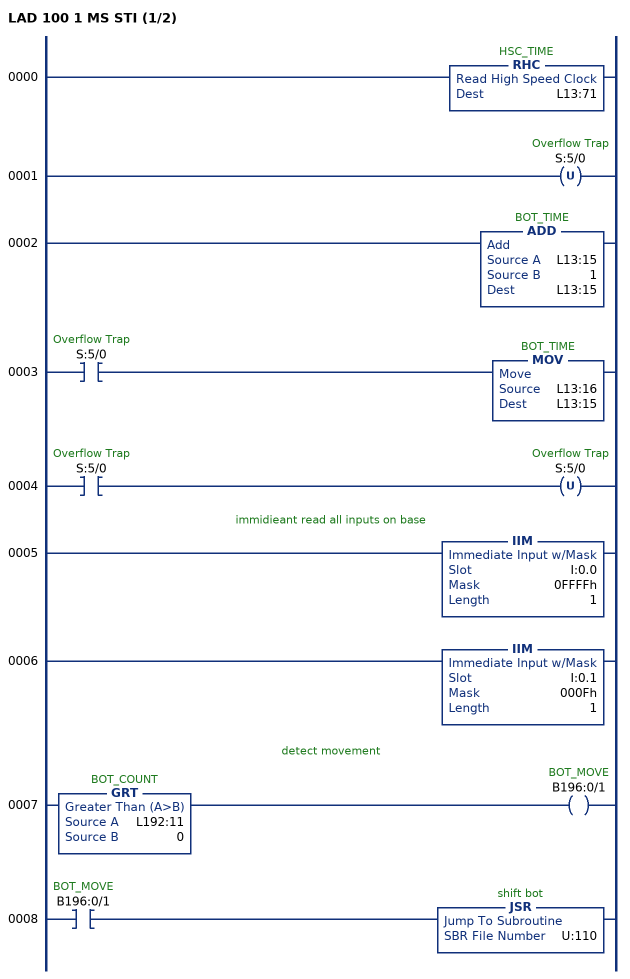
% Rung: 0 %
SOR RHC L13:71 EOR
%   L13:71  HSC_TIME %
% Rung: 1 %
SOR OTU S:5/0 EOR
%   S:5/0  "Overflow Trap" %
% Rung: 2 %
SOR ADD L13:15 1 L13:15 EOR
%   L13:15  BOT_TIME %
% Rung: 3 %
SOR XIC S:5/0 MOV L13:16 L13:15 EOR
%   S:5/0  "Overflow Trap" %
%   L13:16  MIN_LONG %
%   L13:15  BOT_TIME %
% Rung: 4 %
SOR XIC S:5/0 OTU S:5/0 EOR
%   S:5/0  "Overflow Trap" %
% Rung: 5 %
% immidieant read all inputs on base %
SOR IIM I:0.0 0FFFFh 1 EOR
% Rung: 6 %
SOR IIM I:0.1 000Fh 1 EOR
% Rung: 7 %
% detect movement %
SOR GRT L192:11 0 OTE B196:0/1 EOR
%   L192:11  BOT_COUNT %
%   B196:0/1  BOT_MOVE %
% Rung: 8 %
SOR XIC B196:0/1 JSR U:110 EOR
%   B196:0/1  BOT_MOVE %
%   U:110  "shift bot" %

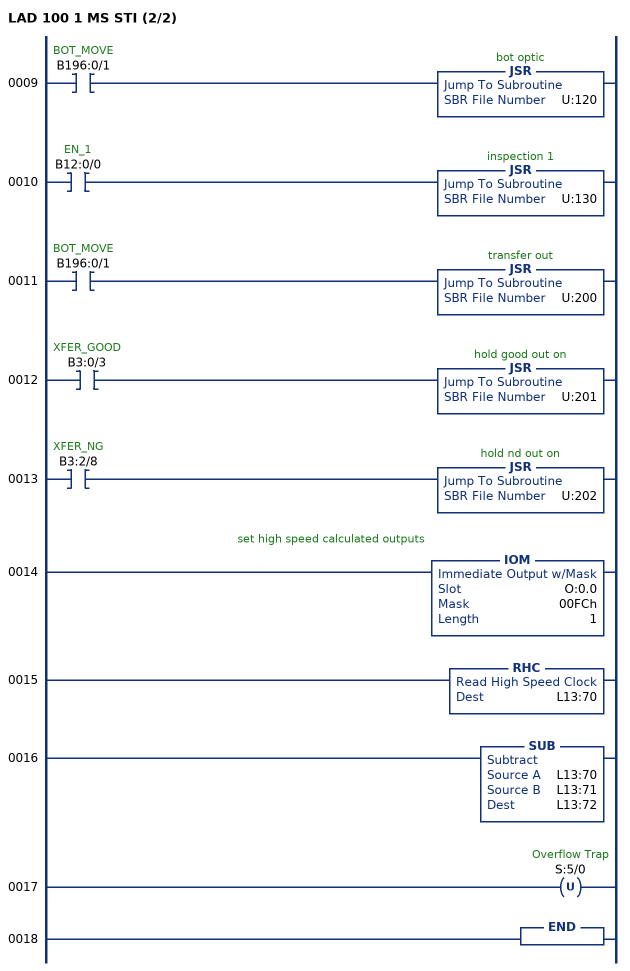
% Rung: 9 %
SOR XIC B196:0/1 JSR U:120 EOR
%   B196:0/1  BOT_MOVE %
%   U:120  "bot optic" %
% Rung: 10 %
SOR XIC B12:0/0 JSR U:130 EOR
%   B12:0/0  EN_1 %
%   U:130  "inspection 1" %
% Rung: 11 %
SOR XIC B196:0/1 JSR U:200 EOR
%   B196:0/1  BOT_MOVE %
%   U:200  "transfer out" %
% Rung: 12 %
SOR XIC B3:0/3 JSR U:201 EOR
%   B3:0/3  XFER_GOOD %
%   U:201  "hold good out on" %
% Rung: 13 %
SOR XIC B3:2/8 JSR U:202 EOR
%   B3:2/8  XFER_NG %
%   U:202  "hold nd out on" %
% Rung: 14 %
% set high speed calculated outputs %
SOR IOM O:0.0 00FCh 1 EOR
% Rung: 15 %
SOR RHC L13:70 EOR
% Rung: 16 %
SOR SUB L13:70 L13:71 L13:72 EOR
%   L13:71  HSC_TIME %
% Rung: 17 %
SOR OTU S:5/0 EOR
%   S:5/0  "Overflow Trap" %
% Rung: 18 %
SOR END EOR

LADDER 102 "SPEED BOT"    % high speed %
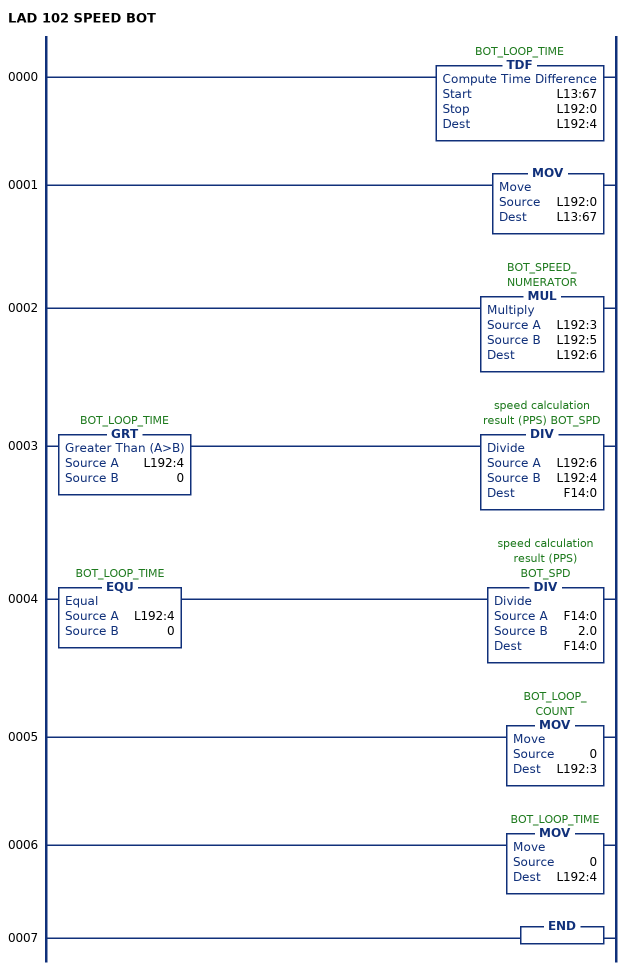
% Rung: 0 %
SOR TDF L13:67 L192:0 L192:4 EOR
%   L192:0  BOT_THIS_TIME  "rtc bot belt movement event time" %
%   L192:4  BOT_LOOP_TIME %
% Rung: 1 %
SOR MOV L192:0 L13:67 EOR
%   L192:0  BOT_THIS_TIME  "rtc bot belt movement event time" %
% Rung: 2 %
SOR MUL L192:3 L192:5 L192:6 EOR
%   L192:3  BOT_LOOP_COUNT %
%   L192:5  TKS_PER_SECOND %
%   L192:6  BOT_SPEED_NUMERATOR %
% Rung: 3 %
SOR GRT L192:4 0 DIV L192:6 L192:4 F14:0 EOR
%   L192:4  BOT_LOOP_TIME %
%   L192:6  BOT_SPEED_NUMERATOR %
%   F14:0  BOT_SPD  "speed calculation result (PPS)" %
% Rung: 4 %
SOR EQU L192:4 0 DIV F14:0 2.0 F14:0 EOR
%   L192:4  BOT_LOOP_TIME %
%   F14:0  BOT_SPD  "speed calculation result (PPS)" %
% Rung: 5 %
SOR MOV 0 L192:3 EOR
%   L192:3  BOT_LOOP_COUNT %
% Rung: 6 %
SOR MOV 0 L192:4 EOR
%   L192:4  BOT_LOOP_TIME %
% Rung: 7 %
SOR END EOR

LADDER 104 "P BOT"    % high speed %
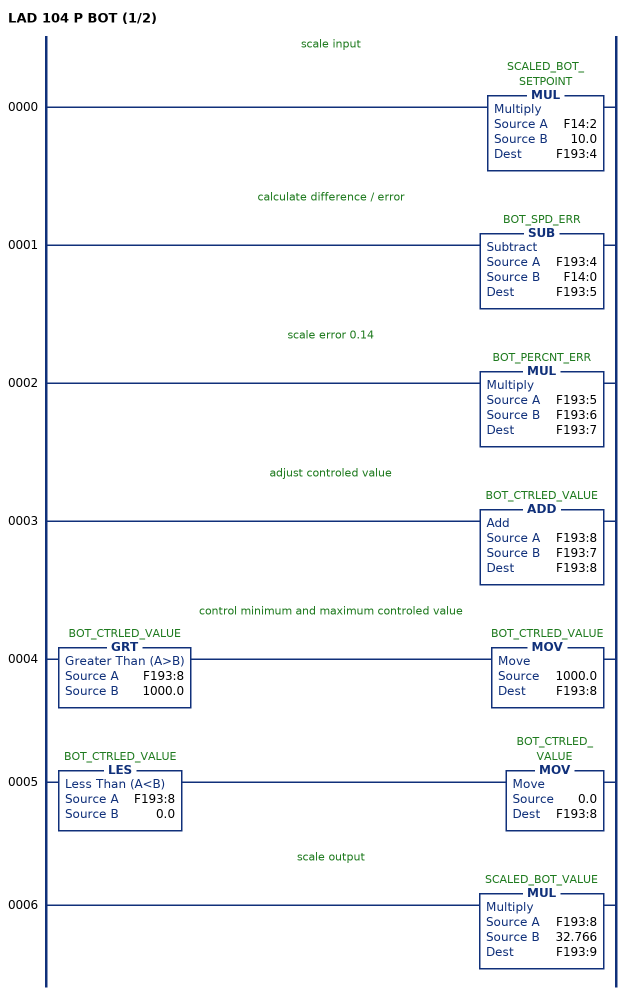
% Rung: 0 %
% scale input %
SOR MUL F14:2 10.0 F193:4 EOR
%   F14:2  BOT_SPD_SETPOINT %
%   F193:4  SCALED_BOT_SETPOINT %
% Rung: 1 %
% calculate difference / error %
SOR SUB F193:4 F14:0 F193:5 EOR
%   F193:4  SCALED_BOT_SETPOINT %
%   F14:0  BOT_SPD  "speed calculation result (PPS)" %
%   F193:5  BOT_SPD_ERR %
% Rung: 2 %
% scale error 0.14 %
SOR MUL F193:5 F193:6 F193:7 EOR
%   F193:5  BOT_SPD_ERR %
%   F193:6  BOT_FDBK_RATIO %
%   F193:7  BOT_PERCNT_ERR %
% Rung: 3 %
% adjust controled value %
SOR ADD F193:8 F193:7 F193:8 EOR
%   F193:8  BOT_CTRLED_VALUE %
%   F193:7  BOT_PERCNT_ERR %
% Rung: 4 %
% control minimum and maximum controled value %
SOR GRT F193:8 1000.0 MOV 1000.0 F193:8 EOR
%   F193:8  BOT_CTRLED_VALUE %
% Rung: 5 %
SOR LES F193:8 0.0 MOV 0.0 F193:8 EOR
%   F193:8  BOT_CTRLED_VALUE %
% Rung: 6 %
% scale output %
SOR MUL F193:8 32.766 F193:9 EOR
%   F193:8  BOT_CTRLED_VALUE %
%   F193:9  SCALED_BOT_VALUE %

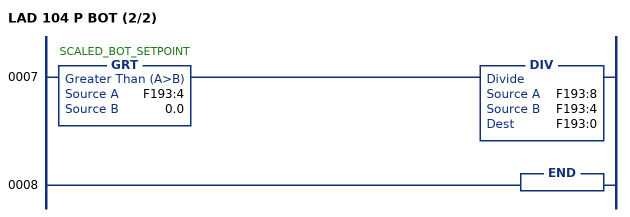
% Rung: 7 %
SOR GRT F193:4 0.0 DIV F193:8 F193:4 F193:0 EOR
%   F193:4  SCALED_BOT_SETPOINT %
%   F193:8  BOT_CTRLED_VALUE %
% Rung: 8 %
SOR END EOR

LADDER 110 "SHIFT BOT"
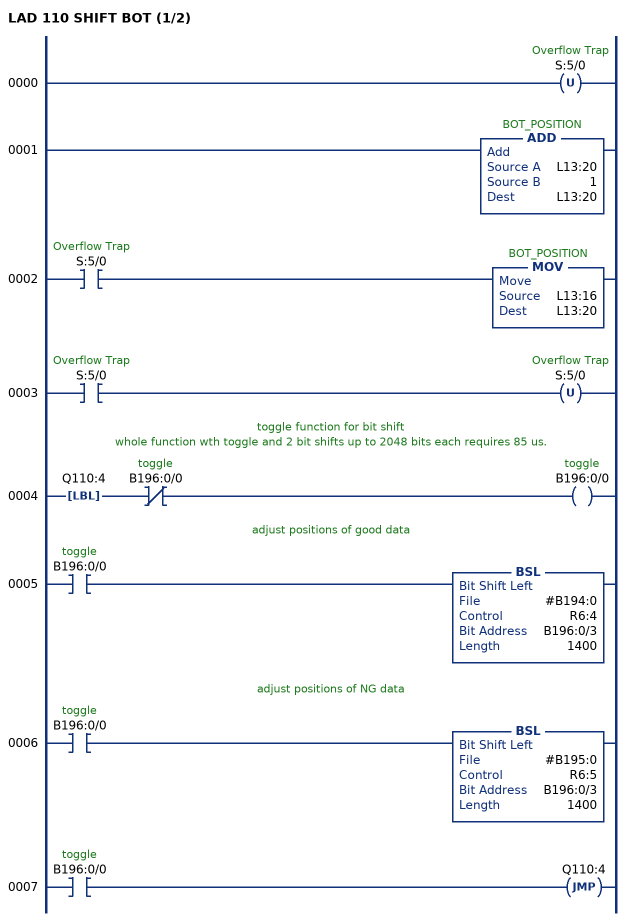
% Rung: 0 %
SOR OTU S:5/0 EOR
%   S:5/0  "Overflow Trap" %
% Rung: 1 %
SOR ADD L13:20 1 L13:20 EOR
%   L13:20  BOT_POSITION %
% Rung: 2 %
SOR XIC S:5/0 MOV L13:16 L13:20 EOR
%   S:5/0  "Overflow Trap" %
%   L13:16  MIN_LONG %
%   L13:20  BOT_POSITION %
% Rung: 3 %
SOR XIC S:5/0 OTU S:5/0 EOR
%   S:5/0  "Overflow Trap" %
% Rung: 4 %
% toggle function for bit shift
% whole function wth toggle and 2 bit shifts up to 2048 bits each requires 85 us. %
SOR LBL Q110:4 XIO B196:0/0 OTE B196:0/0 EOR
%   B196:0/0  "toggle" %
% Rung: 5 %
% adjust positions of good data %
SOR XIC B196:0/0 BSL #B194:0 R6:4 B196:0/3 1400 EOR
%   B196:0/0  "toggle" %
%   B196:0/3  OFF %
% Rung: 6 %
% adjust positions of NG data %
SOR XIC B196:0/0 BSL #B195:0 R6:5 B196:0/3 1400 EOR
%   B196:0/0  "toggle" %
%   B196:0/3  OFF %
% Rung: 7 %
SOR XIC B196:0/0 JMP Q110:4 EOR
%   B196:0/0  "toggle" %

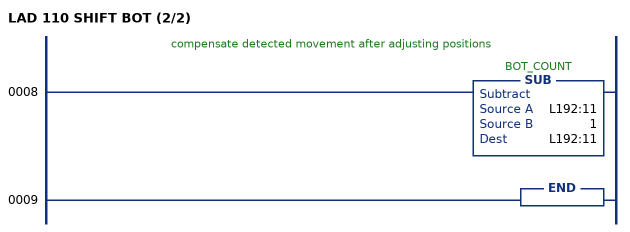
% Rung: 8 %
% compensate detected movement after adjusting positions %
SOR SUB L192:11 1 L192:11 EOR
%   L192:11  BOT_COUNT %
% Rung: 9 %
SOR END EOR

LADDER 120 "BOTOPTIC"
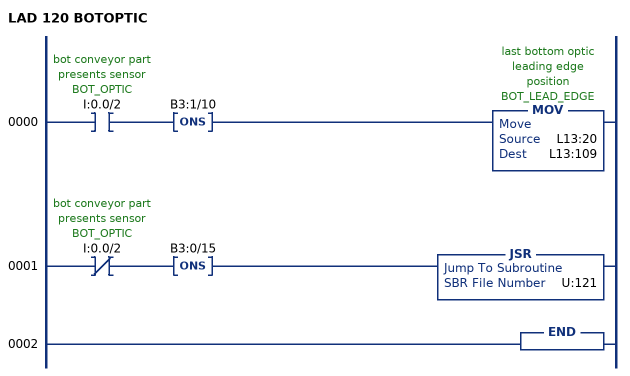
% Rung: 0 %
SOR XIC I:0.0/2 ONS B3:1/10 MOV L13:20 L13:109 EOR
%   I:0.0/2  BOT_OPTIC  "bot conveyor part presents sensor" %
%   L13:20  BOT_POSITION %
%   L13:109  BOT_LEAD_EDGE  "last bottom optic leading edge position" %
% Rung: 1 %
SOR XIO I:0.0/2 ONS B3:0/15 JSR U:121 EOR
%   I:0.0/2  BOT_OPTIC  "bot conveyor part presents sensor" %
% Rung: 2 %
SOR END EOR

LADDER 121 "BOTOPTMES"
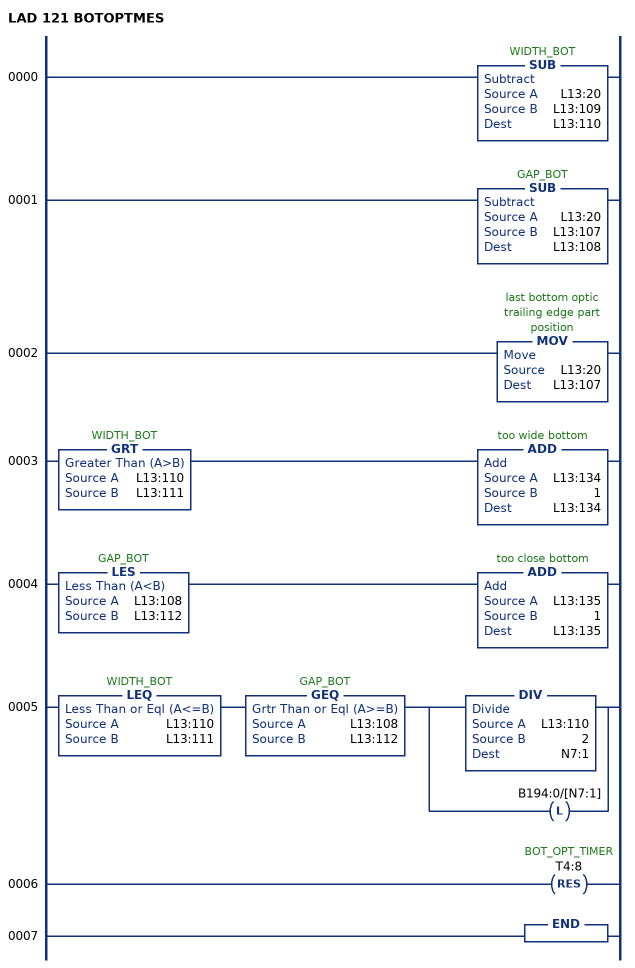
% Rung: 0 %
SOR SUB L13:20 L13:109 L13:110 EOR
%   L13:20  BOT_POSITION %
%   L13:109  BOT_LEAD_EDGE  "last bottom optic leading edge position" %
%   L13:110  WIDTH_BOT %
% Rung: 1 %
SOR SUB L13:20 L13:107 L13:108 EOR
%   L13:20  BOT_POSITION %
%   L13:107  "last bottom optic trailing edge part position" %
%   L13:108  GAP_BOT %
% Rung: 2 %
SOR MOV L13:20 L13:107 EOR
%   L13:20  BOT_POSITION %
%   L13:107  "last bottom optic trailing edge part position" %
% Rung: 3 %
SOR GRT L13:110 L13:111 ADD L13:134 1 L13:134 EOR
%   L13:110  WIDTH_BOT %
%   L13:111  BOT_MAX_WIDTH %
%   L13:134  "too wide bottom" %
% Rung: 4 %
SOR LES L13:108 L13:112 ADD L13:135 1 L13:135 EOR
%   L13:108  GAP_BOT %
%   L13:112  BOT_MIN_GAP %
%   L13:135  "too close bottom" %
% Rung: 5 %
SOR LEQ L13:110 L13:111 GEQ L13:108 L13:112 BST DIV L13:110 2 N7:1 NXB OTL B194:0/[N7:1] BND EOR
%   L13:110  WIDTH_BOT %
%   L13:111  BOT_MAX_WIDTH %
%   L13:108  GAP_BOT %
%   L13:112  BOT_MIN_GAP %
% Rung: 6 %
SOR RES T4:8 EOR
%   T4:8  BOT_OPT_TIMER %
% Rung: 7 %
SOR END EOR

LADDER 130 "INS1"
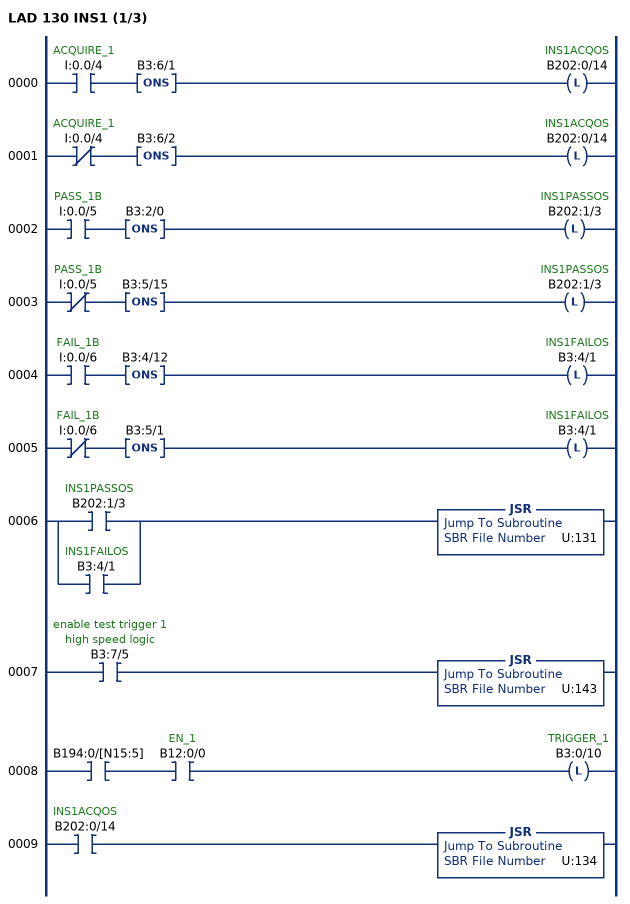
% Rung: 0 %
SOR XIC I:0.0/4 ONS B3:6/1 OTL B202:0/14 EOR
%   I:0.0/4  ACQUIRE_1 %
%   B202:0/14  INS1ACQOS %
% Rung: 1 %
SOR XIO I:0.0/4 ONS B3:6/2 OTL B202:0/14 EOR
%   I:0.0/4  ACQUIRE_1 %
%   B202:0/14  INS1ACQOS %
% Rung: 2 %
SOR XIC I:0.0/5 ONS B3:2/0 OTL B202:1/3 EOR
%   I:0.0/5  PASS_1B %
%   B202:1/3  INS1PASSOS %
% Rung: 3 %
SOR XIO I:0.0/5 ONS B3:5/15 OTL B202:1/3 EOR
%   I:0.0/5  PASS_1B %
%   B202:1/3  INS1PASSOS %
% Rung: 4 %
SOR XIC I:0.0/6 ONS B3:4/12 OTL B3:4/1 EOR
%   I:0.0/6  FAIL_1B %
%   B3:4/1  INS1FAILOS %
% Rung: 5 %
SOR XIO I:0.0/6 ONS B3:5/1 OTL B3:4/1 EOR
%   I:0.0/6  FAIL_1B %
%   B3:4/1  INS1FAILOS %
% Rung: 6 %
SOR BST XIC B202:1/3 NXB XIC B3:4/1 BND JSR U:131 EOR
%   B202:1/3  INS1PASSOS %
%   B3:4/1  INS1FAILOS %
% Rung: 7 %
SOR XIC B3:7/5 JSR U:143 EOR
%   B3:7/5  "enable test trigger 1 high speed logic" %
% Rung: 8 %
SOR XIC B194:0/[N15:5] XIC B12:0/0 OTL B3:0/10 EOR
%   N15:5  INS_1_TRIG_LOC %
%   B12:0/0  EN_1 %
%   B3:0/10  TRIGGER_1 %
% Rung: 9 %
SOR XIC B202:0/14 JSR U:134 EOR
%   B202:0/14  INS1ACQOS %

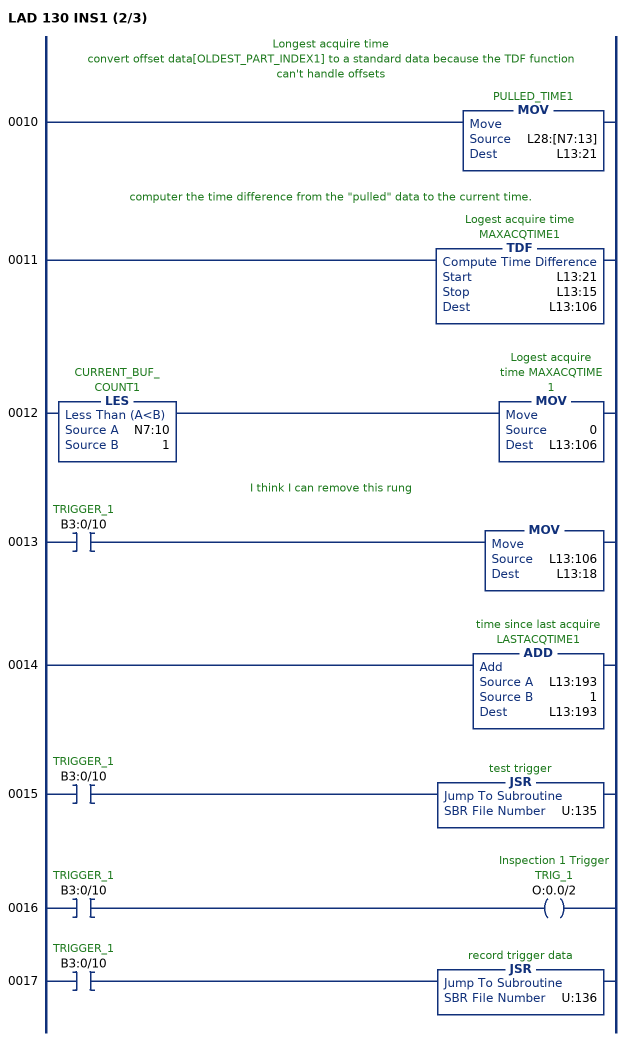
% Rung: 10 %
% Longest acquire time
% convert offset data[OLDEST_PART_INDEX1] to a standard data because the TDF function can't handle offsets %
SOR MOV L28:[N7:13] L13:21 EOR
%   N7:13  OLDEST_PART_INDEX1 %
%   L13:21  PULLED_TIME1 %
% Rung: 11 %
% computer the time difference from the "pulled" data to the current time. %
SOR TDF L13:21 L13:15 L13:106 EOR
%   L13:21  PULLED_TIME1 %
%   L13:15  BOT_TIME %
%   L13:106  MAXACQTIME1  "Logest acquire time" %
% Rung: 12 %
SOR LES N7:10 1 MOV 0 L13:106 EOR
%   N7:10  CURRENT_BUF_COUNT1 %
%   L13:106  MAXACQTIME1  "Logest acquire time" %
% Rung: 13 %
% I think I can remove this rung %
SOR XIC B3:0/10 MOV L13:106 L13:18 EOR
%   B3:0/10  TRIGGER_1 %
%   L13:106  MAXACQTIME1  "Logest acquire time" %
% Rung: 14 %
SOR ADD L13:193 1 L13:193 EOR
%   L13:193  LASTACQTIME1  "time since last acquire" %
% Rung: 15 %
SOR XIC B3:0/10 JSR U:135 EOR
%   B3:0/10  TRIGGER_1 %
%   U:135  "test trigger" %
% Rung: 16 %
SOR XIC B3:0/10 OTE O:0.0/2 EOR
%   B3:0/10  TRIGGER_1 %
%   O:0.0/2  TRIG_1  "Inspection 1 Trigger" %
% Rung: 17 %
SOR XIC B3:0/10 JSR U:136 EOR
%   B3:0/10  TRIGGER_1 %
%   U:136  "record trigger data" %

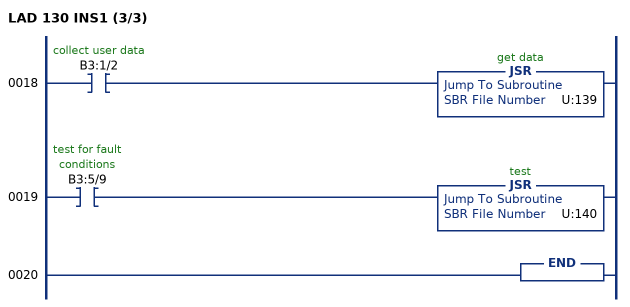
% Rung: 18 %
SOR XIC B3:1/2 JSR U:139 EOR
%   B3:1/2  "collect user data" %
%   U:139  "get data" %
% Rung: 19 %
SOR XIC B3:5/9 JSR U:140 EOR
%   B3:5/9  "test for fault conditions" %
%   U:140  "test" %
% Rung: 20 %
SOR END EOR

LADDER 131 "INS1RESULT"
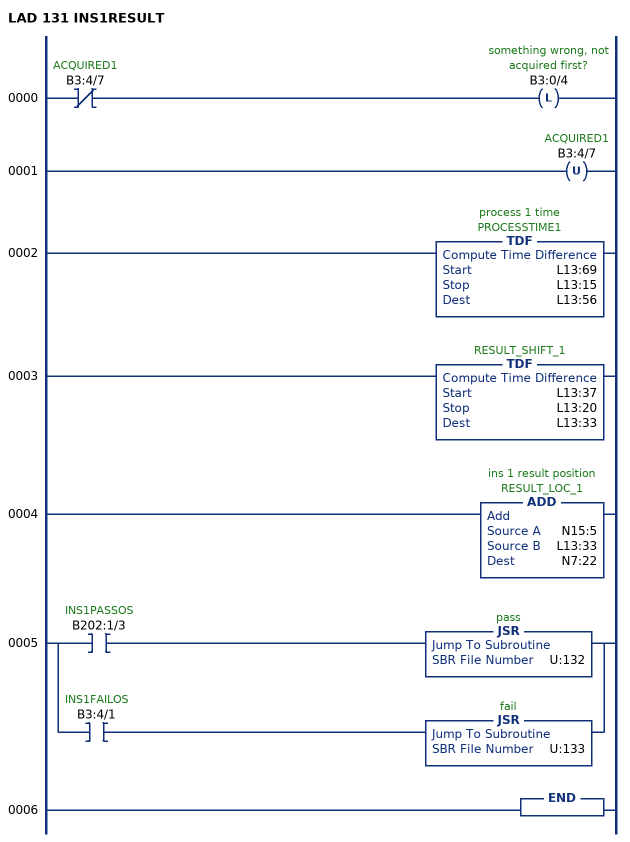
% Rung: 0 %
SOR XIO B3:4/7 OTL B3:0/4 EOR
%   B3:4/7  ACQUIRED1 %
%   B3:0/4  "something wrong, not acquired first?" %
% Rung: 1 %
SOR OTU B3:4/7 EOR
%   B3:4/7  ACQUIRED1 %
% Rung: 2 %
SOR TDF L13:69 L13:15 L13:56 EOR
%   L13:69  TIMEOFACQ1  "the time of the last acquire" %
%   L13:15  BOT_TIME %
%   L13:56  PROCESSTIME1  "process 1 time" %
% Rung: 3 %
SOR TDF L13:37 L13:20 L13:33 EOR
%   L13:37  PROCESS_START_POS_1 %
%   L13:20  BOT_POSITION %
%   L13:33  RESULT_SHIFT_1 %
% Rung: 4 %
SOR ADD N15:5 L13:33 N7:22 EOR
%   N15:5  INS_1_TRIG_LOC %
%   L13:33  RESULT_SHIFT_1 %
%   N7:22  RESULT_LOC_1  "ins 1 result position" %
% Rung: 5 %
SOR BST XIC B202:1/3 JSR U:132 NXB XIC B3:4/1 JSR U:133 BND EOR
%   B202:1/3  INS1PASSOS %
%   U:132  "pass" %
%   B3:4/1  INS1FAILOS %
%   U:133  "fail" %
% Rung: 6 %
SOR END EOR

LADDER 132 "INS1PASS"
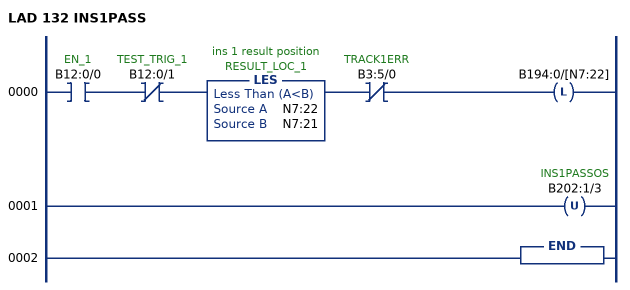
% Rung: 0 %
SOR XIC B12:0/0 XIO B12:0/1 LES N7:22 N7:21 XIO B3:5/0 OTL B194:0/[N7:22] EOR
%   B12:0/0  EN_1 %
%   B12:0/1  TEST_TRIG_1 %
%   N7:22  RESULT_LOC_1  "ins 1 result position" %
%   N7:21  "part shift 1" %
%   B3:5/0  TRACK1ERR %
% Rung: 1 %
SOR OTU B202:1/3 EOR
%   B202:1/3  INS1PASSOS %
% Rung: 2 %
SOR END EOR

LADDER 133 "INS1FAIL"
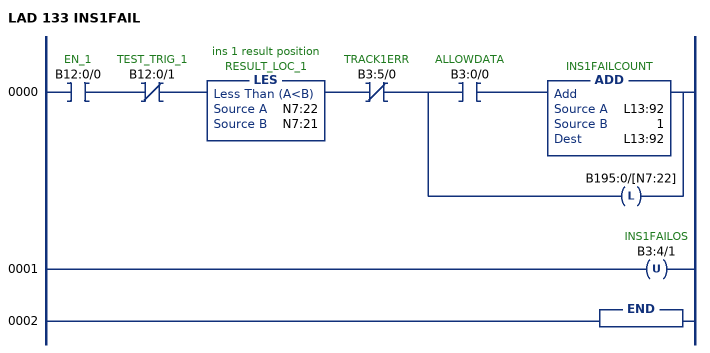
% Rung: 0 %
SOR XIC B12:0/0 XIO B12:0/1 LES N7:22 N7:21 XIO B3:5/0 BST XIC B3:0/0 ADD L13:92 1 L13:92 NXB OTL B195:0/[N7:22] BND EOR
%   B12:0/0  EN_1 %
%   B12:0/1  TEST_TRIG_1 %
%   N7:22  RESULT_LOC_1  "ins 1 result position" %
%   N7:21  "part shift 1" %
%   B3:5/0  TRACK1ERR %
%   B3:0/0  ALLOWDATA %
%   L13:92  INS1FAILCOUNT %
% Rung: 1 %
SOR OTU B3:4/1 EOR
%   B3:4/1  INS1FAILOS %
% Rung: 2 %
SOR END EOR

LADDER 134 "INS1ACQ"
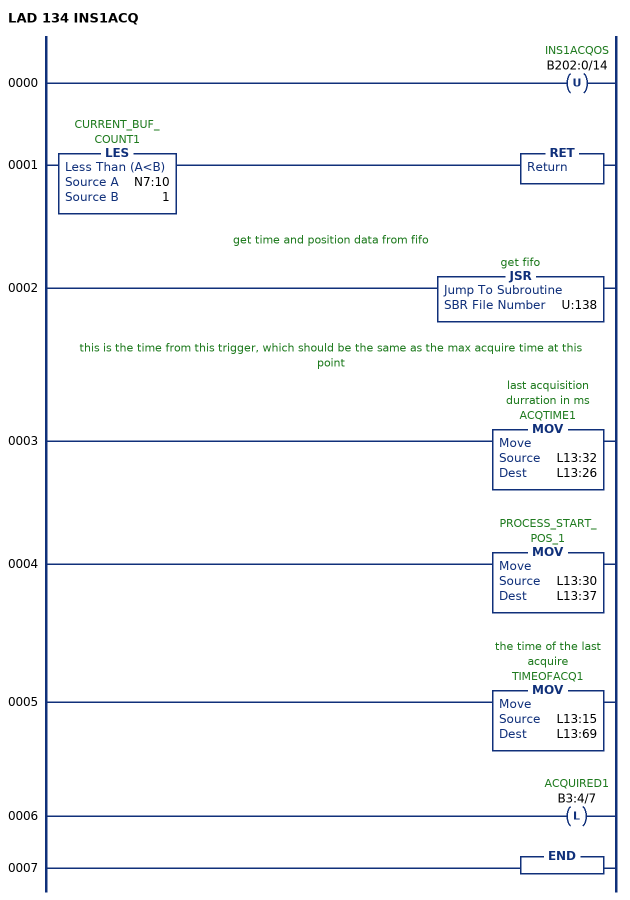
% Rung: 0 %
SOR OTU B202:0/14 EOR
%   B202:0/14  INS1ACQOS %
% Rung: 1 %
SOR LES N7:10 1 RET EOR
%   N7:10  CURRENT_BUF_COUNT1 %
% Rung: 2 %
% get time and position data from fifo %
SOR JSR U:138 EOR
%   U:138  "get fifo" %
% Rung: 3 %
% this is the time from this trigger, which should be the same as the max acquire time at this point %
SOR MOV L13:32 L13:26 EOR
%   L13:32  TIME_SPAN1 %
%   L13:26  ACQTIME1  "last acquisition durration in ms" %
% Rung: 4 %
SOR MOV L13:30 L13:37 EOR
%   L13:30  PULLED_POSITION1 %
%   L13:37  PROCESS_START_POS_1 %
% Rung: 5 %
SOR MOV L13:15 L13:69 EOR
%   L13:15  BOT_TIME %
%   L13:69  TIMEOFACQ1  "the time of the last acquire" %
% Rung: 6 %
SOR OTL B3:4/7 EOR
%   B3:4/7  ACQUIRED1 %
% Rung: 7 %
SOR END EOR

LADDER 135 "Q1TIMETEST"
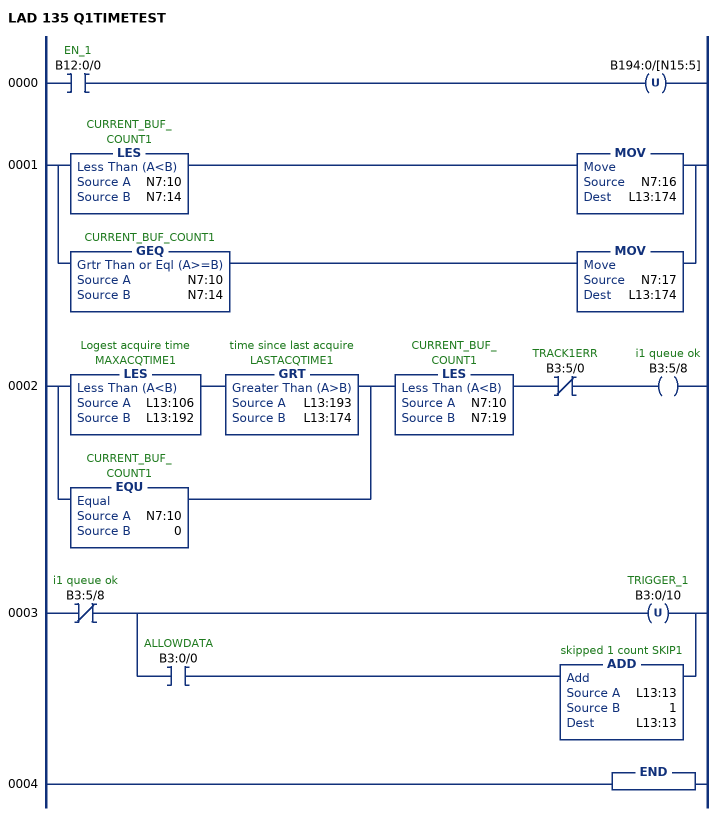
% Rung: 0 %
SOR XIC B12:0/0 OTU B194:0/[N15:5] EOR
%   B12:0/0  EN_1 %
%   N15:5  INS_1_TRIG_LOC %
% Rung: 1 %
SOR BST LES N7:10 N7:14 MOV N7:16 L13:174 NXB GEQ N7:10 N7:14 MOV N7:17 L13:174 BND EOR
%   N7:10  CURRENT_BUF_COUNT1 %
% Rung: 2 %
SOR BST LES L13:106 L13:192 GRT L13:193 L13:174 NXB EQU N7:10 0 BND LES N7:10 N7:19 XIO B3:5/0 OTE B3:5/8 EOR
%   L13:106  MAXACQTIME1  "Logest acquire time" %
%   L13:192  ACQTIMELIMIT1 %
%   L13:193  LASTACQTIME1  "time since last acquire" %
%   N7:10  CURRENT_BUF_COUNT1 %
%   N7:19  "maximum buffers" %
%   B3:5/0  TRACK1ERR %
%   B3:5/8  "i1 queue ok" %
% Rung: 3 %
SOR XIO B3:5/8 BST OTU B3:0/10 NXB XIC B3:0/0 ADD L13:13 1 L13:13 BND EOR
%   B3:5/8  "i1 queue ok" %
%   B3:0/10  TRIGGER_1 %
%   B3:0/0  ALLOWDATA %
%   L13:13  SKIP1  "skipped 1 count" %
% Rung: 4 %
SOR END EOR

LADDER 136 "INS1TRIG"
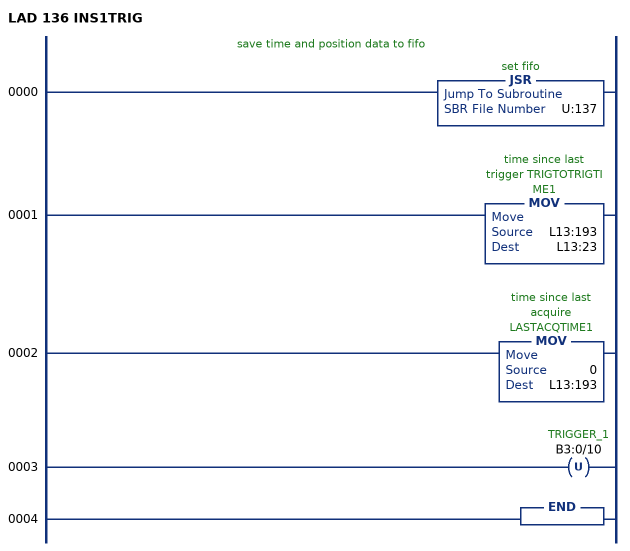
% Rung: 0 %
% save time and position data to fifo %
SOR JSR U:137 EOR
%   U:137  "set fifo" %
% Rung: 1 %
SOR MOV L13:193 L13:23 EOR
%   L13:193  LASTACQTIME1  "time since last acquire" %
%   L13:23  TRIGTOTRIGTIME1  "time since last trigger" %
% Rung: 2 %
SOR MOV 0 L13:193 EOR
%   L13:193  LASTACQTIME1  "time since last acquire" %
% Rung: 3 %
SOR OTU B3:0/10 EOR
%   B3:0/10  TRIGGER_1 %
% Rung: 4 %
SOR END EOR

LADDER 137 "FIFO1SET"
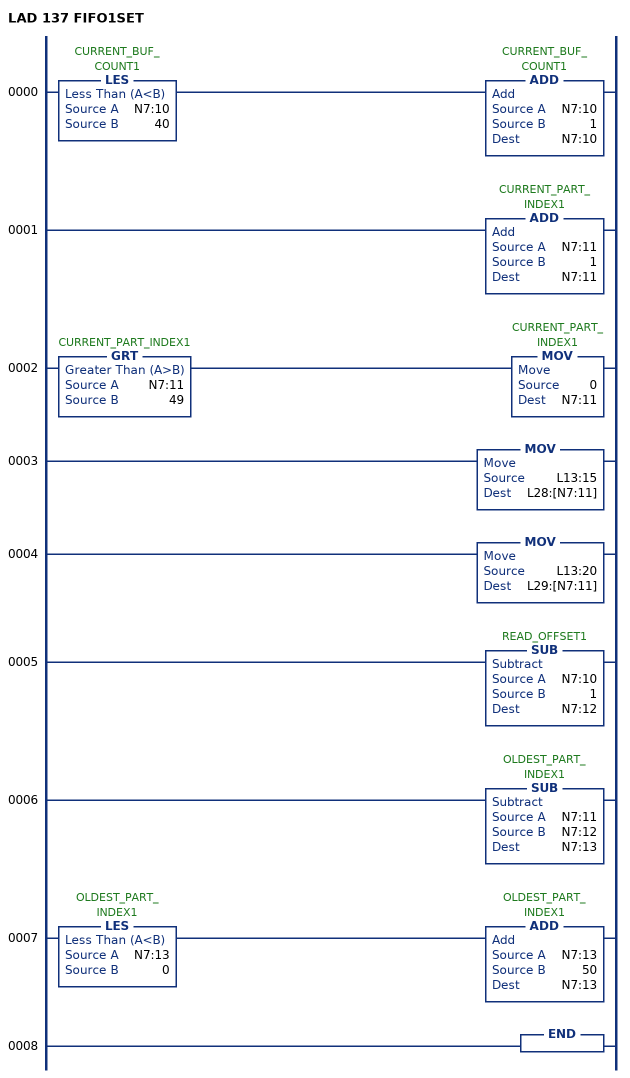
% Rung: 0 %
SOR LES N7:10 40 ADD N7:10 1 N7:10 EOR
%   N7:10  CURRENT_BUF_COUNT1 %
% Rung: 1 %
SOR ADD N7:11 1 N7:11 EOR
%   N7:11  CURRENT_PART_INDEX1 %
% Rung: 2 %
SOR GRT N7:11 49 MOV 0 N7:11 EOR
%   N7:11  CURRENT_PART_INDEX1 %
% Rung: 3 %
SOR MOV L13:15 L28:[N7:11] EOR
%   L13:15  BOT_TIME %
%   N7:11  CURRENT_PART_INDEX1 %
% Rung: 4 %
SOR MOV L13:20 L29:[N7:11] EOR
%   L13:20  BOT_POSITION %
%   N7:11  CURRENT_PART_INDEX1 %
% Rung: 5 %
SOR SUB N7:10 1 N7:12 EOR
%   N7:10  CURRENT_BUF_COUNT1 %
%   N7:12  "READ_OFFSET1" %
% Rung: 6 %
SOR SUB N7:11 N7:12 N7:13 EOR
%   N7:11  CURRENT_PART_INDEX1 %
%   N7:12  "READ_OFFSET1" %
%   N7:13  OLDEST_PART_INDEX1 %
% Rung: 7 %
SOR LES N7:13 0 ADD N7:13 50 N7:13 EOR
%   N7:13  OLDEST_PART_INDEX1 %
% Rung: 8 %
SOR END EOR

LADDER 138 "FIFO1GET"
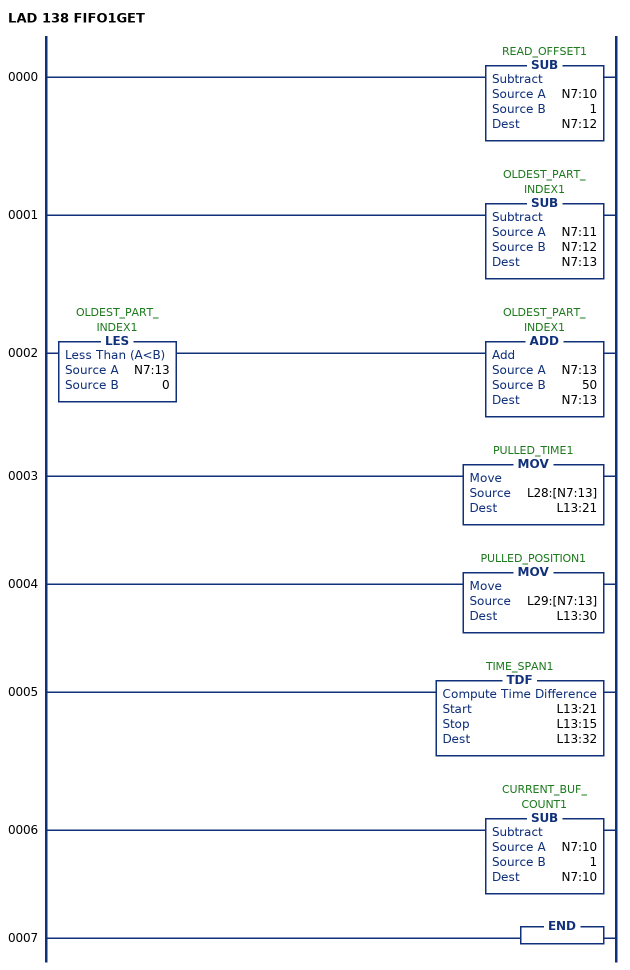
% Rung: 0 %
SOR SUB N7:10 1 N7:12 EOR
%   N7:10  CURRENT_BUF_COUNT1 %
%   N7:12  "READ_OFFSET1" %
% Rung: 1 %
SOR SUB N7:11 N7:12 N7:13 EOR
%   N7:11  CURRENT_PART_INDEX1 %
%   N7:12  "READ_OFFSET1" %
%   N7:13  OLDEST_PART_INDEX1 %
% Rung: 2 %
SOR LES N7:13 0 ADD N7:13 50 N7:13 EOR
%   N7:13  OLDEST_PART_INDEX1 %
% Rung: 3 %
SOR MOV L28:[N7:13] L13:21 EOR
%   N7:13  OLDEST_PART_INDEX1 %
%   L13:21  PULLED_TIME1 %
% Rung: 4 %
SOR MOV L29:[N7:13] L13:30 EOR
%   N7:13  OLDEST_PART_INDEX1 %
%   L13:30  PULLED_POSITION1 %
% Rung: 5 %
SOR TDF L13:21 L13:15 L13:32 EOR
%   L13:21  PULLED_TIME1 %
%   L13:15  BOT_TIME %
%   L13:32  TIME_SPAN1 %
% Rung: 6 %
SOR SUB N7:10 1 N7:10 EOR
%   N7:10  CURRENT_BUF_COUNT1 %
% Rung: 7 %
SOR END EOR

LADDER 139 "INSDATA1"    % used for analysis %
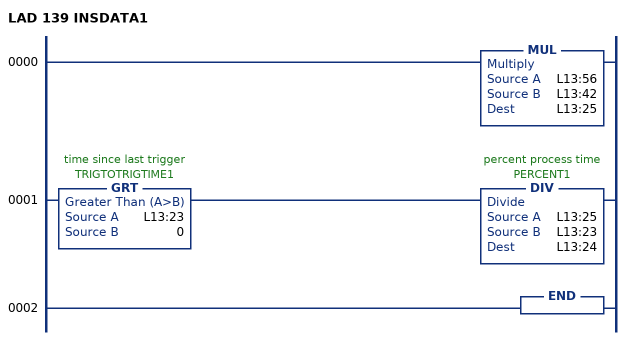
% Rung: 0 %
SOR MUL L13:56 L13:42 L13:25 EOR
%   L13:56  PROCESSTIME1  "process 1 time" %
% Rung: 1 %
SOR GRT L13:23 0 DIV L13:25 L13:23 L13:24 EOR
%   L13:23  TRIGTOTRIGTIME1  "time since last trigger" %
%   L13:24  PERCENT1  "percent process time" %
% Rung: 2 %
SOR END EOR

LADDER 140 "TESTFAULT1"
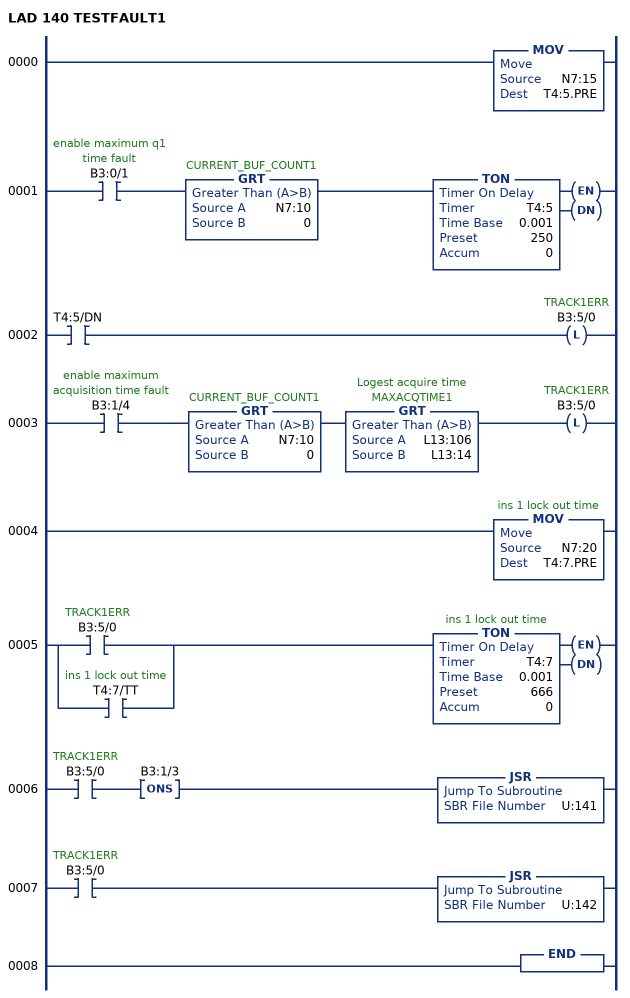
% Rung: 0 %
SOR MOV N7:15 T4:5.PRE EOR
%   N7:15  "max allowed ms time for q to be above 1 if safe fault is used" %
% Rung: 1 %
SOR XIC B3:0/1 GRT N7:10 0 TON T4:5 0.001 250 0 EOR
%   B3:0/1  "enable maximum q1 time fault" %
%   N7:10  CURRENT_BUF_COUNT1 %
% Rung: 2 %
SOR XIC T4:5/DN OTL B3:5/0 EOR
%   B3:5/0  TRACK1ERR %
% Rung: 3 %
SOR XIC B3:1/4 GRT N7:10 0 GRT L13:106 L13:14 OTL B3:5/0 EOR
%   B3:1/4  "enable maximum acquisition time fault" %
%   N7:10  CURRENT_BUF_COUNT1 %
%   L13:106  MAXACQTIME1  "Logest acquire time" %
%   L13:14  "maximum of the longest acquire time allowed if maximum acquire time fault is enabled" %
%   B3:5/0  TRACK1ERR %
% Rung: 4 %
SOR MOV N7:20 T4:7.PRE EOR
%   N7:20  "ms time setting to lock out inspection to give all pending images a chance to clear" %
%   T4:7  "ins 1 lock out time" %
% Rung: 5 %
SOR BST XIC B3:5/0 NXB XIC T4:7/TT BND TON T4:7 0.001 666 0 EOR
%   B3:5/0  TRACK1ERR %
%   T4:7  "ins 1 lock out time" %
% Rung: 6 %
SOR XIC B3:5/0 ONS B3:1/3 JSR U:141 EOR
%   B3:5/0  TRACK1ERR %
% Rung: 7 %
SOR XIC B3:5/0 JSR U:142 EOR
%   B3:5/0  TRACK1ERR %
% Rung: 8 %
SOR END EOR

LADDER 141 "INS1FIX1"
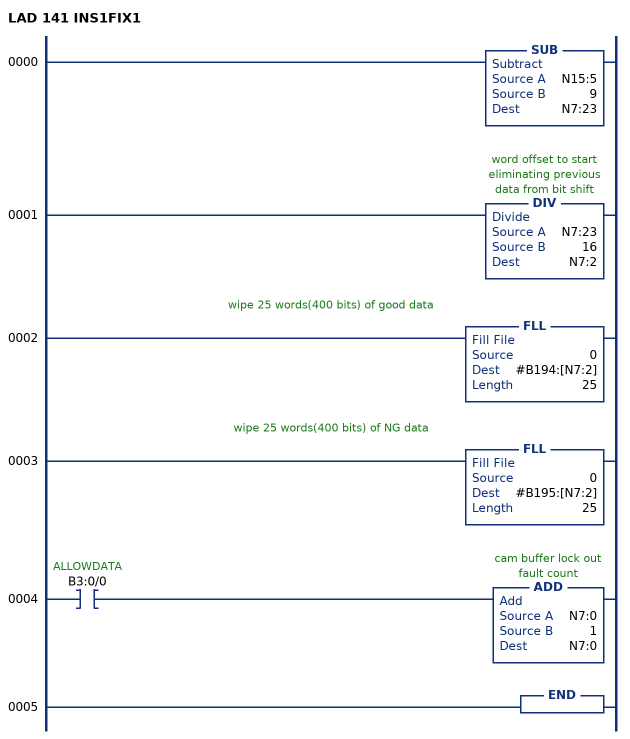
% Rung: 0 %
SOR SUB N15:5 9 N7:23 EOR
%   N15:5  INS_1_TRIG_LOC %
% Rung: 1 %
SOR DIV N7:23 16 N7:2 EOR
%   N7:2  "word offset to start eliminating previous data from bit shift" %
% Rung: 2 %
% wipe 25 words(400 bits) of good data %
SOR FLL 0 #B194:[N7:2] 25 EOR
%   N7:2  "word offset to start eliminating previous data from bit shift" %
% Rung: 3 %
% wipe 25 words(400 bits) of NG data %
SOR FLL 0 #B195:[N7:2] 25 EOR
%   N7:2  "word offset to start eliminating previous data from bit shift" %
% Rung: 4 %
SOR XIC B3:0/0 ADD N7:0 1 N7:0 EOR
%   B3:0/0  ALLOWDATA %
%   N7:0  "cam buffer lock out fault count" %
% Rung: 5 %
SOR END EOR

LADDER 142 "INS1FIX2"
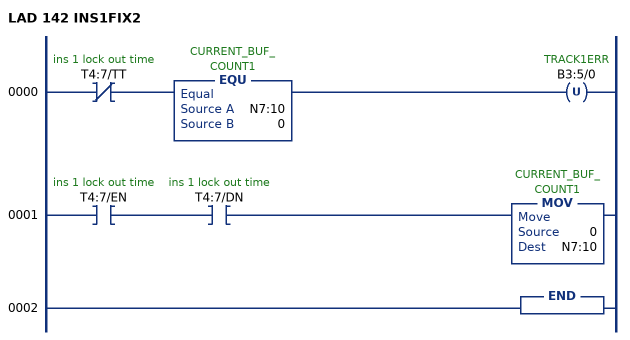
% Rung: 0 %
SOR XIO T4:7/TT EQU N7:10 0 OTU B3:5/0 EOR
%   T4:7  "ins 1 lock out time" %
%   N7:10  CURRENT_BUF_COUNT1 %
%   B3:5/0  TRACK1ERR %
% Rung: 1 %
SOR XIC T4:7/EN XIC T4:7/DN MOV 0 N7:10 EOR
%   T4:7  "ins 1 lock out time" %
%   N7:10  CURRENT_BUF_COUNT1 %
% Rung: 2 %
SOR END EOR

LADDER 143 "HS TRIG1"
